PROGRAM MAIN
VAR
END_VAR

END_PROGRAM

(* stored: Version 1.1.0.1, ProductVersion 3.1.4024.12
   POU MAIN: Id {17eacdce-cfd8-0dc0-36b6-efec9594056c}, SpecialFunc None *)
